// TwinCAT 3 PLC project ArbiterPLC
// Title: LFE-ARBITER
// Company: SLAC - LCLS
// ProjectVersion: 0.0.0
// ProgramVersion: 3.1.4022.7
// CompilerDefines: L
// libraries:
//   PMPS, * (SLAC - LCLS)
//   Tc2_MC2, * (Beckhoff Automation GmbH)
//   Tc2_Standard, * (Beckhoff Automation GmbH)
//   Tc2_System, * (Beckhoff Automation GmbH)
//   Tc2_SystemCX, * (Beckhoff Automation GmbH)
//   Tc2_Utilities, * (Beckhoff Automation GmbH)
//   Tc3_Module, * (Beckhoff Automation GmbH)
//   LCLS General,2.10.0,SLAC
// project tree:
//   / FFOTask.TcTTO (not stored), PlcTask.TcTTO (not stored)
//   GVLs/ GVL.TcGVL, GVL_CheckBounds.TcGVL (not stored)
//   ImplicitChecks/ CheckBounds.TcPOU (not stored), CheckRangeSigned.TcPOU (not stored), CheckRangeUnsigned.TcPOU (not stored)
//   POUs/ CurrentBPUpdate.TcPOU, CXDisplay.TcPOU (not stored), Fast_Faults_Evaluate.TcPOU, MachineSimulation.TcPOU, MAIN.TcPOU, PMPS_Arbiter.TcPOU, P_OpticsProtection.TcPOU, P_SATT.TcPOU, Testing.TcPOU (not stored)
// real-time tasks:
//   TASK PlcTask: cycle T#10ms, priority 2, ADS port 350
//   TASK FFOTask: cycle T#1ms, priority 1, ADS port 351
// I/O:
//   DEVICE Device 1 (EtherCAT), AmsNetId 0.0.0.0.2.1
//     Term 12 (EK1200)
//     Box 23 (CU1128) [CU1128 6x EtherCAT junction]
//       plc-lfe-optics [EL6695 EtherCAT Bridge terminal (Secondary)]
//       plc-lfe-motion [EL6695 EtherCAT Bridge terminal (Secondary)]
//       plc-lfe-vacuum [EL6695 EtherCAT Bridge terminal (Secondary)]
//       plc-lfe-gem [EL6692 EtherCAT Bridge terminal (Secondary)]
//       Term 28 (CU1128-B) [CU1128 6x EtherCAT junction - Dev A]
//         plc-txi-lfe-optics
//       Term 29 (CU1128-C) [CU1128 6x EtherCAT junction - Dev B]
//         plc-txi-lfe-vacuum
//         plc-xrt-homs
//     plc-txi-lfe-motion [EL6695 EtherCAT Bridge terminal (Secondary)]
// variable links:
//   ArbiterPLC Instance <-> Device 1 (EtherCAT)
//     PlcTask Inputs/MAIN.fbEcatDiag.arrEcMasterNetId <-> InfoData/AmsNetId
//     PlcTask Inputs/MAIN.fbEcatDiag.nEcMasterDevState <-> Inputs/DevState
//     PlcTask Inputs/MAIN.fbEcatDiag.nEcMasterDeviceId <-> InfoData/DevId
//     PlcTask Inputs/MAIN.fbEcatDiag.nEcMasterSlaveCount <-> Inputs/SlaveCount
//     PlcTask Inputs/MAIN.fbEcatDiag.nEcMasterSlaveCountCfg <-> InfoData/CfgSlaveCount
//     PlcTask Inputs/MAIN.fbEcatDiag.wFrmXWcState <-> Inputs/Frm1WcState
//   ArbiterPLC Instance <-> Device 1 (EtherCAT)/Box 23 (CU1128)/Term 28 (CU1128-B)/plc-txi-lfe-optics
//     PlcTask Inputs/CurrentBPUpdate.i_MR1L1_ENC <-> IO Inputs/MR1L1_Y_ENC
//     PlcTask Inputs/PMPS_Arbiter.plc_txi_lfe_optics_PMPS_IO.i_Connected <-> SYNC Inputs/External device not connected
//     PlcTask Inputs/PMPS_Arbiter.plc_txi_lfe_optics_PMPS_IO.i_RequestedBP <-> IO Inputs/RequestedBP
//     PlcTask Inputs/PMPS_Arbiter.plc_txi_lfe_optics_PMPS_IO.i_WcState <-> WcState/WcStateIn
//     PlcTask Outputs/PMPS_Arbiter.plc_txi_lfe_optics_PMPS_IO.o_CurrentBP <-> IO Outputs/CurrentBP
//   ArbiterPLC Instance <-> Device 1 (EtherCAT)/Box 23 (CU1128)/Term 29 (CU1128-C)/plc-txi-lfe-vacuum
//     PlcTask Inputs/PMPS_Arbiter.plc_txi_lfe_vacuum_PMPS_IO.i_Connected <-> SYNC Inputs/External device not connected
//     PlcTask Inputs/PMPS_Arbiter.plc_txi_lfe_vacuum_PMPS_IO.i_RequestedBP <-> IO Inputs/RequestedBP
//     PlcTask Inputs/PMPS_Arbiter.plc_txi_lfe_vacuum_PMPS_IO.i_TxPDOState <-> SYNC Inputs/TxPDO state
//     PlcTask Inputs/PMPS_Arbiter.plc_txi_lfe_vacuum_PMPS_IO.i_WcState <-> WcState/WcStateIn
//     PlcTask Outputs/PMPS_Arbiter.plc_txi_lfe_vacuum_PMPS_IO.o_CurrentBP <-> IO Outputs/CurrentBP
//   ArbiterPLC Instance <-> Device 1 (EtherCAT)/Box 23 (CU1128)/Term 29 (CU1128-C)/plc-xrt-homs
//     PlcTask Inputs/PMPS_Arbiter.plc_xrt_homs_PMPS_IO.i_Connected <-> SYNC Inputs/External device not connected
//     PlcTask Inputs/PMPS_Arbiter.plc_xrt_homs_PMPS_IO.i_RequestedBP <-> IO Inputs/RequestedBP
//     PlcTask Inputs/PMPS_Arbiter.plc_xrt_homs_PMPS_IO.i_TxPDOState <-> SYNC Inputs/TxPDO state
//     PlcTask Inputs/PMPS_Arbiter.plc_xrt_homs_PMPS_IO.i_WcState <-> WcState/WcStateIn
//     PlcTask Outputs/PMPS_Arbiter.plc_xrt_homs_PMPS_IO.o_CurrentBP <-> IO Outputs/CurrentBP
//   ArbiterPLC Instance <-> Device 1 (EtherCAT)/Box 23 (CU1128)/plc-lfe-gem
//     PlcTask Inputs/PMPS_Arbiter.plc_lfe_gatt_PMPS_IO.i_Connected <-> SYNC Inputs/External device not connected
//     PlcTask Inputs/PMPS_Arbiter.plc_lfe_gatt_PMPS_IO.i_RequestedBP <-> IO Inputs/RequestedBP
//     PlcTask Inputs/PMPS_Arbiter.plc_lfe_gatt_PMPS_IO.i_TxPDOState <-> SYNC Inputs/TxPDO state
//     PlcTask Inputs/PMPS_Arbiter.plc_lfe_gatt_PMPS_IO.i_WcState <-> WcState/WcStateIn
//     PlcTask Outputs/PMPS_Arbiter.plc_lfe_gatt_PMPS_IO.o_CurrentBP <-> IO Outputs/CurrentBP
//   ArbiterPLC Instance <-> Device 1 (EtherCAT)/Box 23 (CU1128)/plc-lfe-motion
//     PlcTask Inputs/PMPS_Arbiter.plc_lfe_motion_PMPS_IO.i_Connected <-> SYNC Inputs/External device not connected
//     PlcTask Inputs/PMPS_Arbiter.plc_lfe_motion_PMPS_IO.i_RequestedBP <-> IO Inputs/RequestedBP
//     PlcTask Inputs/PMPS_Arbiter.plc_lfe_motion_PMPS_IO.i_TxPDOState <-> SYNC Inputs/TxPDO state
//     PlcTask Inputs/PMPS_Arbiter.plc_lfe_motion_PMPS_IO.i_WcState <-> WcState/WcStateIn
//     PlcTask Inputs/P_SATT.i_SattArrStatus_LFE <-> IO Inputs/SattArrayStatus
//     PlcTask Inputs/P_SATT.i_bWcStateIn_lfe_mot <-> WcState/WcStateIn
//     PlcTask Inputs/P_SATT.i_bWcStateOut_lfe_mot <-> WcState/WcStateOut
//     PlcTask Inputs/P_SATT.i_nState_lfe_mot <-> InfoData/State
//     PlcTask Outputs/PMPS_Arbiter.plc_lfe_motion_PMPS_IO.o_CurrentBP <-> IO Outputs/CurrentBP
//     PlcTask Outputs/P_SATT.q_SattArrayReq <-> IO Outputs/SattArrayReq
//   ArbiterPLC Instance <-> Device 1 (EtherCAT)/Box 23 (CU1128)/plc-lfe-optics
//     PlcTask Inputs/CurrentBPUpdate.i_MR1L0_ENC <-> IO Inputs/MR1L0_Pitch_ENC
//     PlcTask Inputs/PMPS_Arbiter.plc_lfe_optics_PMPS_IO.i_Connected <-> SYNC Inputs/External device not connected
//     PlcTask Inputs/PMPS_Arbiter.plc_lfe_optics_PMPS_IO.i_RequestedBP <-> IO Inputs/RequestedBP
//     PlcTask Inputs/PMPS_Arbiter.plc_lfe_optics_PMPS_IO.i_TxPDOState <-> SYNC Inputs/TxPDO state
//     PlcTask Inputs/PMPS_Arbiter.plc_lfe_optics_PMPS_IO.i_WcState <-> WcState/WcStateIn
//     PlcTask Outputs/PMPS_Arbiter.plc_lfe_optics_PMPS_IO.o_CurrentBP <-> IO Outputs/CurrentBP
//   ArbiterPLC Instance <-> Device 1 (EtherCAT)/Box 23 (CU1128)/plc-lfe-vacuum
//     PlcTask Inputs/PMPS_Arbiter.plc_lfe_vac_PMPS_IO.i_Connected <-> SYNC Inputs/External device not connected
//     PlcTask Inputs/PMPS_Arbiter.plc_lfe_vac_PMPS_IO.i_RequestedBP <-> IO Inputs/RequestedBP
//     PlcTask Inputs/PMPS_Arbiter.plc_lfe_vac_PMPS_IO.i_TxPDOState <-> SYNC Inputs/TxPDO state
//     PlcTask Inputs/PMPS_Arbiter.plc_lfe_vac_PMPS_IO.i_WcState <-> WcState/WcStateIn
//     PlcTask Outputs/PMPS_Arbiter.plc_lfe_vac_PMPS_IO.o_CurrentBP <-> IO Outputs/CurrentBP
//   ArbiterPLC Instance <-> Device 1 (EtherCAT)/Term 12 (EK1200)/E3 (EK1122)/950-101W-R4-MPS-1/MPS_Relay
//     PlcTask Outputs/CurrentBPUpdate.st1l0Watcher.q_StopperIN_Relay <-> Channel 2/ST1L0_RELAY_IN
//     PlcTask Outputs/CurrentBPUpdate.st1l0Watcher.q_StopperOUT_Relay <-> Channel 1/ST1L0_RELAY_OUT
//   ArbiterPLC Instance <-> Device 1 (EtherCAT)/Term 12 (EK1200)/E3 (EK1122)/950-101W-R4-MPS-1/PPS_Stoppers
//     PlcTask Inputs/CurrentBPUpdate.st1l0Watcher.i_StopperInLS <-> Channel 1/ST1L0_PPS_IN
//     PlcTask Inputs/CurrentBPUpdate.st1l1Watcher.i_StopperInLS <-> Channel 3/ST1L1_PPS_IN
//     PlcTask Inputs/CurrentBPUpdate.st1l0Watcher.i_StopperOutLS <-> Channel 2/ST1L0_PPS_OUT
//     PlcTask Inputs/CurrentBPUpdate.st1l1Watcher.i_StopperOutLS <-> Channel 4/ST1L1_PPS_OUT
//   ArbiterPLC Instance <-> Device 1 (EtherCAT)/Term 12 (EK1200)/FFO
//     PlcTask Outputs/GVL.g_FastFaultOutput1.q_xFastFaultOut <-> Channel 1/Output
//     PlcTask Outputs/GVL.g_FastFaultOutput2.q_xFastFaultOut <-> Channel 2/Output
//   ArbiterPLC Instance <-> Device 1 (EtherCAT)/Term 12 (EK1200)/PMPS_Premp
//     PlcTask Outputs/CurrentBPUpdate.st1l1Watcher.q_StopperIN_Relay <-> Channel 6/Output
//     PlcTask Outputs/PMPS_Arbiter.fbCuInterface.q_CLTS_ASSERTION_LINES[1] <-> Channel 9/Output
//     PlcTask Outputs/PMPS_Arbiter.fbCuInterface.q_CLTS_ASSERTION_LINES[2] <-> Channel 10/Output
//     PlcTask Outputs/PMPS_Arbiter.fbCuInterface.q_CLTS_ASSERTION_LINES[3] <-> Channel 11/Output
//     PlcTask Outputs/PMPS_Arbiter.fbMPSInterface.q_BC_ASSERTION_LINES[{1..4}] <-> Channel {1..4}/Output  (4 links)
//   ArbiterPLC Instance <-> Device 1 (EtherCAT)/plc-txi-lfe-motion
//     PlcTask Inputs/PMPS_Arbiter.plc_txi_lfe_motion_PMPS_IO.i_Connected <-> SYNC Inputs/External device not connected
//     PlcTask Inputs/PMPS_Arbiter.plc_txi_lfe_motion_PMPS_IO.i_RequestedBP <-> IO Inputs/RequestedBP
//     PlcTask Inputs/PMPS_Arbiter.plc_txi_lfe_motion_PMPS_IO.i_TxPDOState <-> SYNC Inputs/TxPDO state
//     PlcTask Inputs/PMPS_Arbiter.plc_txi_lfe_motion_PMPS_IO.i_WcState <-> WcState/WcStateIn
//     PlcTask Inputs/PMPS_Arbiter.plc_txi_lfe_optics_PMPS_IO.i_TxPDOState <-> SYNC Inputs/TxPDO state
//     PlcTask Outputs/PMPS_Arbiter.plc_txi_lfe_motion_PMPS_IO.o_CurrentBP <-> IO Outputs/CurrentBP

// ---- GVLs/GVL.TcGVL

VAR_GLOBAL
   {attribute 'pytmc' := '
    pv: @(PREFIX)Arbiter:01
    '}
    g_fbArbiter1	:	FB_Arbiter(25);

    ReqBP	:	ST_BeamParams; //Currently the placeholder for the fully arbitrated BP set

    //Example implementation of the FFO

    {attribute 'pytmc' := '
    pv: @(PREFIX)FFO:01
    '}
    {attribute 'TcLinkTo' := '.q_xFastFaultOut:=TIIB[FFO]^Channel 1^Output'}
    g_FastFaultOutput1	:	FB_HardwareFFOutput := (bAutoReset := TRUE);

    {attribute 'pytmc' := '
    pv: @(PREFIX)FFO:02
    '}
    {attribute 'TcLinkTo' := '.q_xFastFaultOut:=TIIB[FFO]^Channel 2^Output'}
    g_FastFaultOutput2	:	FB_HardwareFFOutput := (bAutoReset := TRUE);

    g_rTestingVelocity	:	LREAL := PMPS_GVL.VISIBLE_TEST_VELOCITY;

    AttemptReset    :   BOOL; // For testing
END_VAR

VAR_GLOBAL CONSTANT
    MAX_FAST_FAULTS : UINT := 100;
END_VAR

// ---- POUs/CurrentBPUpdate.TcPOU
PROGRAM CurrentBPUpdate
VAR
    {attribute 'pytmc' := '
        pv: @(PREFIX)PE
    '}
    fbLPhotonEnergy : FB_LPhotonEnergy;

    {attribute 'pytmc' := '
        pv: @(PREFIX)L:Rate
        link: IOC:BSY0:MP01:BYKIK_RATE
        field: EGU RateEnum
    '}
    fbBYKIK_Rate : FB_LREALFromEPICS := (
        iMaximumValidSeverity := 2);

    {attribute 'pytmc' := '
        pv: @(PREFIX)
    '}
    fbEPICSLRate : FB_RateFromEPICS;

    {attribute 'pytmc' := '
        pv: @(PREFIX)L:BC
        link: SIOC:SYS0:MP03:SC_HXR_BC
        field: EGU BCEnum
    '}
    fbMPS_BeamClass : FB_LREALFromEPICS := (
        iMaximumValidSeverity := 2);

        {attribute 'pytmc' := '
        pv: @(PREFIX)
    '}
    fbEPICSLBeamClass : FB_BeamClassFromEPICS;

    {attribute 'pytmc' := '
        pv: @(PREFIX)L:Mode
        link: SIOC:FEEH:MP01:FACMODE_RBV
    '}
    fbHXR_MachineMode : FB_LREALFromEPICS := (
        iMaximumValidSeverity := 2);

    {attribute 'pytmc' := '
        pv: @(PREFIX)
    '}
    fbEPICSLMachineMode : FB_MachineModeFromEPICS;


    //All Sold attenuators requests are summerrized into this one output
    {attribute 'TcLinkTo' := 'TIIB[plc-lfe-motion]^IO Outputs^rPhotonEnergy'}
    q_rPhotonEnergy AT %Q* : REAL;
    // Stoppers

    {attribute 'TcLinkTo' := '
                .i_StopperInLS:=TIIB[PPS_Stoppers]^Channel 1^ST1L0_PPS_IN;
                .i_StopperOutLS:=TIIB[PPS_Stoppers]^Channel 2^ST1L0_PPS_OUT;
                .q_StopperOUT_Relay:=TIIB[MPS_Relay]^Channel 1^ST1L0_RELAY_OUT;
                .q_StopperIN_Relay:=TIIB[MPS_Relay]^Channel 2^ST1L0_RELAY_IN;
    '}
    st1l0Watcher : FB_LStopper(
        PMPS.L_Stopper.ST1L0,
        'ST1L0');
      {attribute 'TcLinkTo' := '
                .i_StopperInLS:=TIIB[PPS_Stoppers]^Channel 3^ST1L1_PPS_IN;
                .i_StopperOutLS:=TIIB[PPS_Stoppers]^Channel 4^ST1L1_PPS_OUT;
                .q_StopperIN_Relay:=TIIB[PMPS_Premp]^Channel 6^Output;
    '}
    st1l1Watcher : FB_LStopper(
        PMPS.L_Stopper.ST1L1,
        'ST1L1');
     idx : UINT := 1;
    bcBitmask : WORD:=0;
     // MR1L0 Veto
    ////////////////////////
     {attribute 'TcLinkTo' := 'TIIB[plc-lfe-optics]^IO Inputs^MR1L0_Pitch_ENC'}
      i_MR1L0_ENC AT %I* : UDINT; // MR1L0 encoder from the rix optics system
         cMR1L0_TXI_UpperLimit : UDINT := 11116030+500000;
        cMR1L0_TXI_LowerLimit : UDINT := 11116000-500000;
        cMR1L0_L0_UpperLimit : UDINT := 8602330+100000;
        {attribute 'TcLinkTo' := 'TIIB[PMPS_Premp]^Channel 7^MR1L0 TXI'}
        q_MR1L0_TXI AT %Q* : BOOL; // Signal to accel. MPS that MR1L0 is TXI
        fbMR1L0VetoDevice : FB_LVetoDevice(
            eVetoDeviceIN := L_Stopper.MR1L0_TXI,
            eVetoDeviceOUT := L_Stopper.MR1L0_L0,
            sVetoDeviceName := 'MR1L0');

     // MR1L1 Veto
    ////////////////////////
        {attribute 'TcLinkTo' := 'TIIB[plc-txi-lfe-optics]^IO Inputs^MR1L1_Y_ENC'}
        i_MR1L1_ENC AT %I* : UDINT; // MR1L1 encoder from the rix optics system
        cMR1L1_IN_UpperLimit : UDINT := 108500000;
        cMR1L1_IN_LowerLimit : UDINT := 108600000;
        cMR1L1_OUT_UpperLimit : UDINT := 9100000;// estimated
        {attribute 'TcLinkTo' := 'TIIB[PMPS_Premp]^Channel 8^MR1L1 IN'}
        q_MR1L1_VETO AT %Q* : BOOL; // Signal to accel. MPS that MR1L1 is in
        fbMR1L1VetoDevice : FB_LVetoDevice(
            eVetoDeviceIN := L_Stopper.MR1L1_IN,
            eVetoDeviceOUT := L_Stopper.MR1L1_OUT,
            sVetoDeviceName := 'MR1L1');
END_VAR

// Acquiring photon energy
fbLPhotonEnergy(BP:=PMPS_GVL.stCurrentBeamParameters);

q_rPhotonEnergy := LREAL_TO_REAL(fbLPhotonEnergy.fbHgvpu.fCurrentPhotonEnergy);
//Update current photon energy
PMPS_GVL.stCurrentBeamParameters.neV := LREAL_TO_REAL(fbLPhotonEnergy.fbHgvpu.fCurrentPhotonEnergy);


// Acquiring L-line rate
fbEPICSLRate(BP:=PMPS_GVL.stCurrentBeamParameters, fbBYKIK_Rate:=fbBYKIK_Rate, FFO:=GVL.g_FastFaultOutput1);


// Acquiring L-line BeamClass
fbEPICSLBeamClass(BP:=PMPS_GVL.stCurrentBeamParameters, fbMPS_BeamClass:=fbMPS_BeamClass, FFO:=GVL.g_FastFaultOutput1);

// Acquiring L-line Machine Mode
fbEPICSLMachineMode(BP:=PMPS_GVL.stCurrentBeamParameters, fbMPS_MachineMode:=fbHXR_MachineMode, FFO:=GVL.g_FastFaultOutput1);



// Watching and relaying stopper statuses
st1l0Watcher(stCurrentBP := PMPS_GVL.stCurrentBeamParameters);
st1l1Watcher(stCurrentBP := PMPS_GVL.stCurrentBeamParameters);

// MR1L0 Veto
////////////////////////
   fbMR1L0VetoDevice(
        i_bIn := cMR1L0_TXI_LowerLimit < i_MR1L0_ENC	AND i_MR1L0_ENC < cMR1L0_TXI_UpperLimit,
        i_bOut := i_MR1L0_ENC < cMR1L0_L0_UpperLimit,
        q_bIN => q_MR1L0_TXI,
        stCurrentBP:= PMPS_GVL.stCurrentBeamParameters);


// MR1L1 Veto
////////////////////////
   fbMR1L1VetoDevice(
        i_bIn := cMR1L1_IN_LowerLimit < i_MR1L1_ENC	AND i_MR1L1_ENC < cMR1L1_IN_UpperLimit,
        i_bOut := i_MR1L1_ENC < cMR1L1_OUT_UpperLimit,
        q_bIN => q_MR1L1_VETO,
        stCurrentBP:= PMPS_GVL.stCurrentBeamParameters);

END_PROGRAM

// ---- POUs/Fast_Faults_Evaluate.TcPOU
PROGRAM Fast_Faults_Evaluate
VAR
END_VAR

//g_FastFaultOutput1.EvaluateOutput(bAutoReset:=TRUE);
//g_FastFaultOutput2.EvaluateOutput(bAutoReset:=TRUE);

// FF
//g_FastFaultOutput1.Execute();
//g_FastFaultOutput2.Execute();

END_PROGRAM

// ---- POUs/MachineSimulation.TcPOU
PROGRAM MachineSimulation
VAR
    fbMachine	:	FB_MachineSimulator; //Simulates attenuator as well
    fbeVSimulator : FB_eVSimulator := (NoiseLevel := 1);
    rTestPhotonEnergy : REAL;
END_VAR

// reV Simulator
fbeVSimulator();

// Machine simulator
fbMachine(
    i_stAssertedParams := PMPS_GVL.stRequestedBeamParameters,
    iq_stMachineParams := PMPS_GVL.stCurrentBeamParameters,
    i_xFault	:= NOT GVL.g_FastFaultOutput1.q_xFastFaultOut,
    xEnableAtt := TRUE,
    xEnableRate := FALSE,
    xEnablePE := TRUE
    );

//PMPS_GVL.stCurrentBeamParameters.neVRange := F_eVRangeCalculator(rTestPhotonEnergy, PMPS_GVL.stCurrentBeamParameters.neVRange);
//PMPS_GVL.stCurrentBeamParameters.neVRange := 0;

END_PROGRAM

// ---- POUs/MAIN.TcPOU
PROGRAM MAIN
VAR
    Initialize	:	BOOL := TRUE;

    fbLogHandler : FB_LogHandler;
    fbEcatDiag : FB_EcatDiagWrapper;

    idx: UINT;

    //System Time
     {attribute 'pytmc' := '
        pv: @(PREFIX)SystemDT
        io: i
     '}
    SystemTime:DINT;
    fbTime : FB_LocalSystemTime := ( bEnable := TRUE, dwCycle := 1 ); //Get current system time, used for override
    fbTime_to_UTC: FB_TzSpecificLocalTimeToSystemTime;
    fbGetTimeZone: FB_GetTimeZoneInformation;
END_VAR

//Arbiter PLC

IF Initialize THEN
    Initialize := FALSE;

    // Setting apertures to zero for now
    FOR idx := 1 TO PMPS_GVL.MAX_APERTURES DO
        PMPS_GVL.stCurrentBeamParameters.astApertures[idx].Height := 0;
        PMPS_GVL.stCurrentBeamParameters.astApertures[idx].Width := 0;
    END_FOR
END_IF

// Ethercat Diagnostics
fbEcatDiag();

CurrentBPUpdate();

///////////////////////////////////////////////////
// This code should be disabled or removed in deployment
// Might have a switch to change to simulation mode
MachineSimulation();
//Testing();
///////////////////////////////////////////////////

// PMPS Functionality

PMPS_Arbiter();
A_SystemTime();

P_SATT();

fbLogHandler();

P_OpticsProtection();

//FF
g_FastFaultOutput1.Execute();
g_FastFaultOutput2.Execute();

ACTION A_SystemTime:
//Get local System Time
fbTime(sNetID:='');
//Get Time Zone
fbGetTimeZone(sNetID:='',bExecute:=TRUE,tTimeout:=T#10S);
//change local time to UTC to be compatible with unix time epoch widget
fbTime_to_UTC(in:= fbTime.systemTime , tzInfo:=fbGetTimeZone.tzInfo);

SystemTime:= TO_DINT(TO_DT(SystemTime_TO_DT(fbTime_to_UTC.out)));
END_ACTION

ACTION Initialize:

END_ACTION

END_PROGRAM

// ---- POUs/PMPS_Arbiter.TcPOU
PROGRAM PMPS_Arbiter
VAR

    fbBPRequestor : FB_BPRequestor; // Updates global PMPS RequestedBeamParams
    {attribute 'pytmc' := '
    pv: @(PREFIX)PhotonEnergyWatcher
    '}
    fbPhotonEnergyWatcher	:	FB_PhotonEnergyWatcher;
    {attribute 'pytmc' := '
    pv: @(PREFIX)BeamClassWatcher
    '}
    fbBeamClassWatcher : FB_BeamClassWatcher;
    {attribute 'pytmc' := '
    pv: @(PREFIX)BeamClassOutputs
    '}
    fbMPSInterface	:	FB_BeamClassOutputs_BCD;
    {attribute 'pytmc' := '
    pv: @(PREFIX)CuRateOutputs
    '}
    fbCuInterface	:	FB_CTLS_Outputs;

    {attribute 'pytmc' := '
        pv: @(PREFIX)BeamParamCntl
    '}
    fbBPControl : FB_BPControlDevice(nID:=10);

    (* Subsystem requests use this FB and a pragma link to pass their requests to the arbiter.
    The fb is called on each cycle and updates the arbiter with the current BP set requested
    from the subsystem PLC.*)
    //<TODO> make this so it does input and output to the IF
    (*{attribute 'pytmc' := '
    pv: @(PREFIX):PLC1
    '}*)
    {attribute 'TcLinkTo' := '.i_RequestedBP:=TIIB[plc-lfe-motion]^IO Inputs^RequestedBP;
                                .o_CurrentBP:=TIIB[plc-lfe-motion]^IO Outputs^CurrentBP;
                                .i_Connected:=TIIB[plc-lfe-motion]^SYNC Inputs^External device not connected;
                                .i_WcState:=TIIB[plc-lfe-motion]^WcState^WcStateIn;
                                .i_TxPDOState:=TIIB[plc-lfe-motion]^SYNC Inputs^TxPDO state;
                                '}
    plc_lfe_motion_PMPS_IO : FB_ArbiterToSubSys_IO := (RequestingSystemID := 16#FF0F);

        {attribute 'TcLinkTo' := '.i_RequestedBP:=TIIB[plc-lfe-optics]^IO Inputs^RequestedBP;
                                .o_CurrentBP:=TIIB[plc-lfe-optics]^IO Outputs^CurrentBP;
                                .i_Connected:=TIIB[plc-lfe-optics]^SYNC Inputs^External device not connected;
                                .i_WcState:=TIIB[plc-lfe-optics]^WcState^WcStateIn;
                                .i_TxPDOState:=TIIB[plc-lfe-optics]^SYNC Inputs^TxPDO state;
                                '}
    plc_lfe_optics_PMPS_IO : FB_ArbiterToSubSys_IO := (RequestingSystemID := 16#FF10);

        {attribute 'TcLinkTo' := '.i_RequestedBP:=TIIB[plc-xrt-homs]^IO Inputs^RequestedBP;
                                .o_CurrentBP:=TIIB[plc-xrt-homs]^IO Outputs^CurrentBP;
                                .i_Connected:=TIIB[plc-xrt-homs]^SYNC Inputs^External device not connected;
                                .i_WcState:=TIIB[plc-xrt-homs]^WcState^WcStateIn;
                                .i_TxPDOState:=TIIB[plc-xrt-homs]^SYNC Inputs^TxPDO state;
                                '}
    plc_xrt_homs_PMPS_IO : FB_ArbiterToSubSys_IO := (RequestingSystemID := 16#FF13);


    {attribute 'TcLinkTo' := '.i_RequestedBP:=TIIB[plc-lfe-vacuum]^IO Inputs^RequestedBP;
                                .o_CurrentBP:=TIIB[plc-lfe-vacuum]^IO Outputs^CurrentBP;
                                .i_Connected:=TIIB[plc-lfe-vacuum]^SYNC Inputs^External device not connected;
                                .i_WcState:=TIIB[plc-lfe-vacuum]^WcState^WcStateIn;
                                .i_TxPDOState:=TIIB[plc-lfe-vacuum]^SYNC Inputs^TxPDO state;
                                '}
    plc_lfe_vac_PMPS_IO : FB_ArbiterToSubSys_IO := (RequestingSystemID := 16#FF11);

        {attribute 'TcLinkTo' := '.i_RequestedBP:=TIIB[plc-lfe-gem]^IO Inputs^RequestedBP;
                                .o_CurrentBP:=TIIB[plc-lfe-gem]^IO Outputs^CurrentBP;
                                .i_Connected:=TIIB[plc-lfe-gem]^SYNC Inputs^External device not connected;
                                .i_WcState:=TIIB[plc-lfe-gem]^WcState^WcStateIn;
                                .i_TxPDOState:=TIIB[plc-lfe-gem]^SYNC Inputs^TxPDO state;
                                '}
    plc_lfe_gatt_PMPS_IO : FB_ArbiterToSubSys_IO := (RequestingSystemID := 16#FF12);



     {attribute 'TcLinkTo' := '.i_RequestedBP:=TIIB[plc-txi-lfe-vacuum]^IO Inputs^RequestedBP;
                                .o_CurrentBP:=TIIB[plc-txi-lfe-vacuum]^IO Outputs^CurrentBP;
                                .i_Connected:=TIIB[plc-txi-lfe-vacuum]^SYNC Inputs^External device not connected;
                                .i_WcState:=TIIB[plc-txi-lfe-vacuum]^WcState^WcStateIn;
                                .i_TxPDOState:=TIIB[plc-txi-lfe-vacuum]^SYNC Inputs^TxPDO state;
                                '}
    plc_txi_lfe_vacuum_PMPS_IO : FB_ArbiterToSubSys_IO := (RequestingSystemID := 16#FF14);

     {attribute 'TcLinkTo' := '.i_RequestedBP:=TIIB[plc-txi-lfe-motion]^IO Inputs^RequestedBP;
                                .o_CurrentBP:=TIIB[plc-txi-lfe-motion]^IO Outputs^CurrentBP;
                                .i_Connected:=TIIB[plc-txi-lfe-motion]^SYNC Inputs^External device not connected;
                                .i_WcState:=TIIB[plc-txi-lfe-motion]^WcState^WcStateIn;
                                .i_TxPDOState:=TIIB[plc-txi-lfe-motion]^SYNC Inputs^TxPDO state;
                                '}
    plc_txi_lfe_motion_PMPS_IO : FB_ArbiterToSubSys_IO := (RequestingSystemID := 16#FF15);

     {attribute 'TcLinkTo' := '.i_RequestedBP:=TIIB[plc-txi-lfe-optics]^IO Inputs^RequestedBP;
                                .o_CurrentBP:=TIIB[plc-txi-lfe-optics]^IO Outputs^CurrentBP;
                                .i_Connected:=TIIB[plc-txi-lfe-optics]^SYNC Inputs^External device not connected;
                                .i_WcState:=TIIB[plc-txi-lfe-optics]^WcState^WcStateIn;
                                .i_TxPDOState:=TIIB[plc-txi-lfe-motion]^SYNC Inputs^TxPDO state;
                                '}
    plc_txi_lfe_optics_PMPS_IO : FB_ArbiterToSubSys_IO := (RequestingSystemID := 16#FF16);

    fbSetPE	:	PE_Ranges;

END_VAR



////////////////////////////////////////////////////////////

// Dummy device for controling pmps beam parameters
fbBPControl(Arbiter:=g_fbArbiter1);

// Updating arbiter with subsystem requests.
// FEE LFE
plc_lfe_motion_PMPS_IO(Arbiter:=GVL.g_fbArbiter1, fbFFHWO:=GVL.g_FastFaultOutput1, Reset:=GVL.AttemptReset, sName:= 'LFE MOTION');
plc_lfe_optics_PMPS_IO(Arbiter:=GVL.g_fbArbiter1, fbFFHWO:=GVL.g_FastFaultOutput1, Reset:=GVL.AttemptReset , sName:= 'LFE OPTICS');
plc_lfe_vac_PMPS_IO(Arbiter:=GVL.g_fbArbiter1, fbFFHWO:=GVL.g_FastFaultOutput1, Reset:=GVL.AttemptReset, sName:= 'LFE VACUUM');
plc_lfe_gatt_PMPS_IO(Arbiter:=GVL.g_fbArbiter1, fbFFHWO:=GVL.g_FastFaultOutput1, Reset:=GVL.AttemptReset, sName:= 'LFE GEMS');
// TXI LFE
plc_txi_lfe_vacuum_PMPS_IO(Arbiter:=GVL.g_fbArbiter1, fbFFHWO:=GVL.g_FastFaultOutput1, Reset:=GVL.AttemptReset, sName:= 'TXI LFE VACUUM');
plc_txi_lfe_motion_PMPS_IO(Arbiter:=GVL.g_fbArbiter1, fbFFHWO:=GVL.g_FastFaultOutput1, Reset:=GVL.AttemptReset, sName:= 'TXI LFE MOTION');
plc_txi_lfe_optics_PMPS_IO(Arbiter:=GVL.g_fbArbiter1, fbFFHWO:=GVL.g_FastFaultOutput1, Reset:=GVL.AttemptReset, sName:= 'TXI LFE OPTICS');
//XRT
plc_xrt_homs_PMPS_IO(Arbiter:=GVL.g_fbArbiter1, fbFFHWO:=GVL.g_FastFaultOutput1, Reset:=GVL.AttemptReset, sName:= 'XRT OPTICS');

//Overriding the preemptive requests from the optics systems until they are valid
//GVL.g_fbArbiter1.RemoveRequest(nReqId:=plc_lfe_optics_PMPS_IO.RequestingSystemID);

// Beam parameter requestor
fbBPRequestor(Arbiter:=GVL.g_fbArbiter1, q_ReqBP => PMPS_GVL.stRequestedBeamParameters);

// Request beam class
fbMPSInterface(BP := PMPS_GVL.stRequestedBeamParameters);

// Request Cu beam rate
fbCuInterface(BP := PMPS_GVL.stRequestedBeamParameters);

// Keep an eye on the beam class
fbBeamClassWatcher(i_stCurrentBeamParams	:= PMPS_GVL.stCurrentBeamParameters,
                    i_stRequestedBeamParams := PMPS_GVL.stRequestedBeamParameters,
                    io_fbFFHWO:= GVL.g_FastFaultOutput1,
                    i_xAutoReset := GVL.AttemptReset);

// Keep an eye on the photon energy
fbPhotonEnergyWatcher(i_stCurrentBeamParams	:= PMPS_GVL.stCurrentBeamParameters,
                    i_stRequestedBeamParams := PMPS_GVL.stRequestedBeamParameters,
                    io_fbFFHWO:= GVL.g_FastFaultOutput1,
                    i_xReset := GVL.AttemptReset);

END_PROGRAM

// ---- POUs/P_SATT.TcPOU
PROGRAM P_SATT
VAR
    //All Solid attenuators requests are summarized into this one output
    {attribute 'TcLinkTo' := 'TIIB[plc-lfe-motion]^IO Outputs^SattArrayReq'}
    q_SattArrayReq AT %Q* : ARRAY [1..PMPS_GVL.AUX_ATTENUATORS] OF ST_PMPS_Attenuator_IO; // Transmission request to ALL PLCs
    //Per PLC current satt trans
    {attribute 'TcLinkTo' := 'TIIB[plc-lfe-motion]^IO Inputs^SattArrayStatus'}
    i_SattArrStatus_LFE AT %I* : ARRAY [1..PMPS_GVL.AUX_ATTENUATORS] OF ST_PMPS_Attenuator_IO; // Transmission status from LFE MOT PLC

    // plc-lfe-motion interface diagnostics
    {attribute 'TcLinkTo' := 'TIIB[plc-lfe-motion]^WcState^WcStateOut'}
    i_bWcStateOut_lfe_mot AT %I* : BOOL;
    {attribute 'TcLinkTo' := 'TIIB[plc-lfe-motion]^WcState^WcStateIn'}
    i_bWcStateIn_lfe_mot AT %I* : BOOL;
    {attribute 'TcLinkTo' := 'TIIB[plc-lfe-motion]^InfoData^State'}
    i_nState_lfe_mot AT %I* : UINT;

    //FFO Connection per PLC
    ffLfeConnection : FB_FastFault := (
        i_DevName := 'PMPS Arbiter',
        i_Desc := 'EtherCAT interface watcher, for lfe-mot connection to systems for attenuation requests. Very rare. Make a note, and if it can be reset, go ahead.',
        i_TypeCode := 16#5);

END_VAR



// Send request from this arbiter to all satts
MEMCPY( ADR(q_SattArrayReq) , ADR(PMPS_GVL.stRequestedBeamParameters.astAttenuators) , PMPS_GVL.AUX_ATTENUATORS * SIZEOF(ST_PMPS_Attenuator_IO) );

//TMO motion PLC SATT current trans update
IF i_bWcStateIn_lfe_mot = 0 AND i_bWcStateOut_lfe_mot = 0 AND i_nState_lfe_mot = 8 THEN
    // 	Recieve current transmission of the satt
    //PMPS_GVL.stCurrentBeamParameters.astAttenuators[PMPS.L_Attenuators.AT2L0].nTran :=  i_SattArrStatus_LFE[PMPS.L_Attenuators.AT2L0].nTran;
    //PMPS_GVL.stCurrentBeamParameters.astAttenuators[PMPS.L_Attenuators.AT2L0].xAttOK :=  i_SattArrStatus_LFE[PMPS.L_Attenuators.AT2L0].xAttOK;
    ffLfeConnection.i_xOK := TRUE;
ELSE
    // Fast fault
    fflfeConnection.i_xOK := FALSE;
END_IF
ffLfeConnection(io_fbFFHWO := g_FastFaultOutput1);

END_PROGRAM

// ---- POUs/P_OpticsProtection.TcPOU
PROGRAM P_OpticsProtection
VAR

    fbFF    :    FB_FastFault :=(
        i_DevName := 'LFE OPTICS',
        i_Desc := 'Fault occurs when MR1L0 is in L0 State and MR1L1 in IN.',
        i_TypeCode := 16#404 );
END_VAR



fbFF(i_xOK := NOT(PMPS.PMPS_GVL.stCurrentBeamParameters.aVetoDevices[PMPS.L_Stopper.MR1L0_L0]
                    AND PMPS.PMPS_GVL.stCurrentBeamParameters.aVetoDevices[PMPS.L_Stopper.MR1L1_IN]),
        io_fbFFHWO :=GVL.g_FastFaultOutput1 , i_xAutoReset := );

END_PROGRAM
